FUNCTION_BLOCK FB_AutoDemo
VAR_INPUT
	bExecute : BOOL;
END_VAR
VAR_OUTPUT
	bBusy : BOOL;
END_VAR
VAR
	nCurStep					: UDINT;
	i							: UDINT;
	nCurRunCount				: UDINT;
	fbMoveDirectAbs				: MC_MoveDirectAbsolute;
	fbMoveLinAbs 				: ARRAY [1..3] OF MC_MoveLinearAbsolute;
	fVeloM						: REAL := 2.0;
	fVeloPer					: REAL := 100.0;
	fAccM						: REAL := 2.3;
	fAccPer						: REAL := 100;
	
	stPrePos					: E6POS;
	stCoordSys					: COORDSYS;
	stApo1						: APO;
	
	fbKRC_Interrupt				: KRC_Interrupt;
	fbKRC_Continue				: KRC_Continue;
	
	iPosCount					: UINT :=1;
END_VAR
VAR CONSTANT
	POSARRLENGTH : UINT := 4;
END_VAR

CASE nCurStep OF
0:
	bBusy := FALSE;

	
	IF bExecute THEN
		iPosCount := 1;
		stApo1.CP_MODE := 0;
		stApo1.CDIS := 0;
		
		FOR i:= 1 TO 2  DO
			fbMoveLinAbs[i](Execute:= FALSE); 
		END_FOR
		fbMoveDirectAbs(Execute:= FALSE); 
		bBusy := TRUE;
		//PTP
		nCurStep := nCurStep + 10;
		nCurRunCount := 0;
		i := 0;
	END_IF
	
10:	
	M_MoveDirectToInitPos();
20:
	fbMoveLinAbs[2]();
	fbMoveLinAbs[3]();
	IF fbMoveLinAbs[1].ComAcpt AND NOT fbMoveLinAbs[2].Busy THEN
		fbMoveLinAbs[1].Execute := FALSE;
		iPosCount := iPosCount + 1;
		IF iPosCount > POSARRLENGTH THEN
			iPosCount := 1;
		END_IF
		nCurStep := nCurStep + 10;
	ELSE
		fbMoveLinAbs[1].Execute := TRUE;
	END_IF
	
	fbMoveLinAbs[1](
			AxisGroupIdx:= GVL.nAxisIndex, 
			Position:= GVL.aPosArray[iPosCount].E6POS, 
			Velocity:= fVeloM, 
			Acceleration:=fAccM , 
			CoordinateSystem:= stCoordSys, 
			OriType:= , 
			Approximate:= stApo1, 
			QueueMode:= 2 , 
			ComAcpt=> , 
			ComBusy=> , 
			Busy=> , 
			Active=> , 
			Done=> , 
			CommandAborted=> , 
			Error=> , 
			ErrorID=> );
		
		
	IF bExecute = FALSE THEN
		nCurStep := 100;
	END_IF

30:	
	fbMoveLinAbs[1]();
	fbMoveLinAbs[3]();
	
	IF fbMoveLinAbs[2].ComAcpt AND NOT fbMoveLinAbs[3].Busy THEN
		fbMoveLinAbs[2].Execute := FALSE;
		iPosCount := iPosCount + 1;
		IF iPosCount > POSARRLENGTH THEN
			iPosCount := 1;
		END_IF
		nCurStep := nCurStep + 10;
	ELSE
		fbMoveLinAbs[2].Execute := TRUE;
	END_IF	
	
	fbMoveLinAbs[2](
		AxisGroupIdx:= gvl.nAxisIndex, 
		Position:= GVL.aPosArray[iPosCount].E6POS, 
		Velocity:= fVeloM, 
		Acceleration:=fAccM , 
		CoordinateSystem:= stCoordSys, 
		OriType:= , 
		Approximate:= stApo1, 
		QueueMode:= 2 , 
		ComAcpt=> , 
		ComBusy=> , 
		Busy=> , 
		Active=> , 
		Done=> , 
		CommandAborted=> , 
		Error=> , 
		ErrorID=> );
		
	
	
	IF bExecute = FALSE THEN
		nCurStep := 100;
	END_IF
	
40:	
	fbMoveLinAbs[1]();
	fbMoveLinAbs[2]();
	
	IF fbMoveLinAbs[3].ComAcpt AND NOT fbMoveLinAbs[1].Busy THEN
		fbMoveLinAbs[3].Execute := FALSE;
		iPosCount := iPosCount + 1;
		IF iPosCount > POSARRLENGTH THEN
			iPosCount := 1;
		END_IF
		nCurStep := 20;
	ELSE
		fbMoveLinAbs[3].Execute := TRUE;
	END_IF	
	
	fbMoveLinAbs[3](
		AxisGroupIdx:= gvl.nAxisIndex, 
		Position:= GVL.aPosArray[iPosCount].E6POS, 
		Velocity:= fVeloM, 
		Acceleration:=fAccM , 
		CoordinateSystem:= stCoordSys, 
		OriType:= , 
		Approximate:= stApo1, 
		QueueMode:= 2 , 
		ComAcpt=> , 
		ComBusy=> , 
		Busy=> , 
		Active=> , 
		Done=> , 
		CommandAborted=> , 
		Error=> , 
		ErrorID=> );
		
	
	
	IF bExecute = FALSE THEN
		nCurStep := 100;
	END_IF
	
100:
	fbMoveLinAbs[1]();
	fbMoveLinAbs[2]();
	fbMoveLinAbs[3]();
	
	IF NOT bExecute AND NOT fbMoveDirectAbs.Busy 
		AND NOT fbMoveLinAbs[1].Busy AND NOT fbMoveLinAbs[2].Busy AND NOT fbMoveLinAbs[3].Busy THEN
		nCurStep := 0;
	END_IF
		
END_CASE

fbKRC_Interrupt(
	AxisGroupIdx:= GVL.nAxisIndex, 
	Execute:= , 
	Fast:= , 
	BrakeActive=> , 
	Error=> , 
	ErrorID=> );
	
fbKRC_Continue(AxisGroupIdx:= GVL.nAxisIndex, Enable:= , Error=> , ErrorID=> );

METHOD M_MoveDirectToInitPos : BOOL
VAR_INPUT
END_VAR
stPrePos := GVL.aPosArray[1].E6POS;
stCoordSys := GVL.aPosArray[1].COORDSYS;

fbMoveDirectAbs(
	AxisGroupIdx:= GVL.nAxisIndex , 
	Execute:= TRUE, 
	Position:= stPrePos, 
	Velocity:= fVeloPer , 
	Acceleration:=fAccPer , 
	CoordinateSystem:= stCoordSys , 
	Approximate:=stApo1 , 
	QueueMode:=  2, 
	ComAcpt=> , 
	ComBusy=> , 
	Busy=> , 
	Active=> , 
	Done=> , 
	CommandAborted=> , 
	Error=> , 
	ErrorID=> );
	
IF fbMoveDirectAbs.Done THEN
	fbMoveDirectAbs(Execute := FALSE); 
	nCurStep := nCurStep + 10;
END_IF
END_METHOD

END_FUNCTION_BLOCK

(* stored: Version 1.1.0.1, ProductVersion 3.1.4024.10
   POU FB_AutoDemo: Id {6cd759e3-5147-48aa-a8e1-fd16d7148084}, SpecialFunc None
   Method M_MoveDirectToInitPos: Id {8a07c01f-60ab-4744-8b98-69965a044512} *)
